PROGRAM MAIN
VAR
	// Variables to call the axis
	AXIS_X		: Master_Axis;
	Axis_is_enabled	: BOOL;
	
	//Variables for axis Home
	Ref	: BOOL;
	Axis_is_at_Home : BOOL;
	
	
END_VAR

AXIS_X ();

AXIS_X.Enable();

IF AXIS_X.Enable() THEN
	Axis_is_enabled := TRUE;
END_IF



//IF Ref THEN
// 	AXIS_X.Home();

//	IF AXIS_X.Home() THEN
//	Axis_is_at_Home := TRUE;	
//	END_IF
	
//END_IF

END_PROGRAM

(* stored: Version 1.1.0.1, ProductVersion 3.1.4024.10
   POU MAIN: Id {6160b492-81c1-4c2c-860a-e8e871705101}, SpecialFunc None *)
